(* IEC 61131-3 sources: repolevel_ST_code_completion/dataset/project_code/卷绕机/FUN, 4 files *)

(* ---- FB_DualAxisEmergencyStop.st ---- *)
FUNCTION_BLOCK FB_DualAxisEmergencyStop
VAR_IN_OUT
	AxisM			:	AXIS_REF_SM3;		// 主轴引用
	AxisS			:	AXIS_REF_SM3;		// 从轴引用
END_VAR
VAR_INPUT
	bExecute		:	BOOL;				// 执行紧急停止
	rDeceleration	:	LREAL := 36000;		// 减速度
END_VAR
VAR_OUTPUT
	bDone			:	BOOL;				// 停止完成
	bBusy			:	BOOL;				// 停止进行中
	bError			:	BOOL;				// 错误标志
END_VAR
VAR
	fbHaltM			:	MC_Halt;			// 主轴停止功能块
	fbHaltS			:	MC_Halt;			// 从轴停止功能块
	fbRtrigExecute	:	R_TRIG;				// 执行上升沿检测
	nState			:	BYTE;				// 内部状态机
END_VAR

fbRtrigExecute(CLK := bExecute);

CASE nState OF
	0: // 空闲/初始化
		bDone := FALSE;
		bBusy := FALSE;
		bError := FALSE;
		fbHaltM(Axis := AxisM, Execute := FALSE);
		fbHaltS(Axis := AxisS, Execute := FALSE);

		IF fbRtrigExecute.Q THEN
			nState := 1;
			bBusy := TRUE;
		END_IF

	1: // 执行双轴停止
		fbHaltM(
			Axis := AxisM,
			Execute := TRUE,
			Deceleration := rDeceleration
		);

		fbHaltS(
			Axis := AxisS,
			Execute := TRUE,
			Deceleration := rDeceleration
		);

		// 等待两轴都停止完成
		IF fbHaltM.Done AND fbHaltS.Done THEN
			nState := 2;
		END_IF

		// 错误检查
		IF fbHaltM.Error OR fbHaltS.Error THEN
			bError := TRUE;
			nState := 100;
		END_IF

	2: // 复位Halt功能块
		fbHaltM(Axis := AxisM, Execute := FALSE);
		fbHaltS(Axis := AxisS, Execute := FALSE);
		nState := 3;

	3: // 完成
		bDone := TRUE;
		bBusy := FALSE;
		nState := 0;

	100: // 错误状态
		bError := TRUE;
		bBusy := FALSE;
		fbHaltM(Execute := FALSE);
		fbHaltS(Execute := FALSE);
		// 等待bExecute复位
		IF NOT bExecute THEN
			nState := 0;
		END_IF
END_CASE

(* ---- FB_DualAxisPower.st ---- *)
FUNCTION_BLOCK FB_DualAxisPower
VAR_IN_OUT
	AxisM		:	AXIS_REF_SM3;		// 主轴引用
	AxisS		:	AXIS_REF_SM3;		// 从轴引用
END_VAR
VAR_INPUT
	bPowerOn	:	BOOL;				// 电源使能信号
END_VAR
VAR_OUTPUT
	bReady		:	BOOL;				// 两轴都准备就绪
	bAxisMReady	:	BOOL;				// 主轴准备状态
	bAxisSReady	:	BOOL;				// 从轴准备状态
	bError		:	BOOL;				// 错误标志
END_VAR
VAR
	fbPowerM	:	SM3_Basic.MC_Power;	// 主轴电源控制
	fbPowerS	:	SM3_Basic.MC_Power;	// 从轴电源控制
END_VAR

// 主轴电源控制
fbPowerM(
	Axis := AxisM,
	Enable := TRUE,
	bRegulatorOn := bPowerOn,
	bDriveStart := bPowerOn
);

// 从轴电源控制
fbPowerS(
	Axis := AxisS,
	Enable := TRUE,
	bRegulatorOn := bPowerOn,
	bDriveStart := bPowerOn
);

// 更新输出状态
bAxisMReady := fbPowerM.Status;
bAxisSReady := fbPowerS.Status;
bReady := fbPowerM.Status AND fbPowerS.Status;

// 错误处理
bError := fbPowerM.Error OR fbPowerS.Error;

(* ---- SeekHome.st ---- *)
FUNCTION_BLOCK SeekHome
VAR_IN_OUT
	_Axis	:	AXIS_REF_SM3;
END_VAR
VAR_INPUT
	_xHome	:	BOOL;
	_xAbort	:	BOOL;
	_nHomeMode	:	HomeMode;
	_fFastHomeVel	:	LREAL;
	_fSlowHomeVel	:	LREAL;
	_fHomeAcc		:	LREAL;
	_fHomeDec		:	LREAL;
	_fHomePos		:	LREAL;
	_xReferenceSwitch	:	BOOL;//typically is true
	_nDirection	:	MC_DIRECTION;
	_xIndexPulse	:	BOOL;
END_VAR
VAR_OUTPUT
	_xBusy	:	BOOL;
	_xDone	:	BOOL;
	_xErr	:	BOOL;
	_iErrId	:	DINT;
END_VAR
VAR
	_fbMoveVel	:	MC_MoveVelocity;
	_fbMoveAbs	:	MC_MoveAbsolute;
	_fbHalt		:	MC_Halt;
	_fbSetPos	:	MC_SetPosition;
	_fbRtrig		:	R_TRIG;
	_fbFtrig		:	F_TRIG;
	_nBDirection	:	MC_DIRECTION;
	_fTempPos		:	LREAL;
	_nState		:	USINT;
	fbRtrig	:	R_TRIG;
END_VAR

//check left / arrive the ReferenceSwitch
_fbRtrig(CLK := _xReferenceSwitch);
_fbFtrig(CLK := _xReferenceSwitch);
fbRtrig(CLK := _xHome);

IF NOT _xHome THEN
	_fbMoveVel(Axis := _Axis,Execute := FALSE);
	_fbMoveAbs(Axis := _Axis,Execute := FALSE);
	_fbHalt(Axis := _Axis,Execute := FALSE);
	_fbSetPos(Axis := _Axis,Execute := FALSE);
	_xDone := FALSE;
	_xErr := FALSE;
END_IF

CASE _nState OF
	0:
		IF fbRtrig.Q THEN
			_xBusy := TRUE;
			_xDone := FALSE;
			_xErr := FALSE;
			_iErrId := 0;

			CASE _nDirection OF //cal which is the invert direction
				MC_DIRECTION.positive:
					_nBDirection := MC_DIRECTION.negative;
				MC_DIRECTION.negative:
					_nBDirection := MC_DIRECTION.positive;
				ELSE
					_xErr := TRUE;
			END_CASE

			CASE _nHomeMode OF
				HomeMode.FAST_ZERO:
					_fTempPos := 0;
					_nState := 21;
				HomeMode.FAST_BSLOW_STOP_S:
					_nState := 1;
				HomeMode.FAST_SLOW_STOP_S:
					_nState := 11;
				HomeMode.FAST_BSLOW_I_STOP_S:
					_nState := 31;
				HomeMode.FAST_SLOW_I_STOP_S:
					_nState := 41;
			END_CASE
		END_IF
	50:
		_fbMoveAbs(Execute := TRUE,Axis := _Axis,Position := _fTempPos,Velocity := _fSlowHomeVel,Acceleration := _fHomeAcc,Deceleration := _fHomeDec);
		IF _fbMoveAbs.Done THEN
			_fbMoveAbs(Execute := FALSE,Axis := _Axis);
			_nState := 100;
		END_IF
		IF _fbMoveAbs.Error THEN//meet error
			_nState := 200;
			_iErrId := _fbMoveAbs.ErrorID;
		END_IF
	100:
		_fbSetPos(Execute := TRUE,Axis := _Axis,Position := _fHomePos,Mode := FALSE);//set absolute position
		IF _fbSetPos.Done THEN
			_fbSetPos(Execute := FALSE,Axis := _Axis);
			_xDone := TRUE;
			_xBusy := FALSE;
			_nState := 0;
		END_IF
		IF _fbSetPos.Error THEN//meet error
			_iErrId := _fbSetPos.ErrorID;
			_nState := 200;
		END_IF
	200:
		_xErr := TRUE;
		_xBusy := FALSE;
		_nState := 0;
END_CASE

FAST_ZERO();
FAST_BSLOW_STOP_S();
FAST_SLOW_STOP_S();
FAST_BSLOW_I_STOP_S();
FAST_SLOW_I_STOP_S();

(* ---- StarWork.st ---- *)
FUNCTION_BLOCK StarWork
VAR_IN_OUT
	_AxisW	:	AXIS_REF_SM3;
	_AxisU	:	AXIS_REF_SM3;
	_AxisV	:	AXIS_REF_SM3;
END_VAR
VAR_INPUT
	_bStart	:	BOOL;
	_bStop	:	BOOL;
	_bCheckR	:	BOOL;
	_bFFlag		:	BOOL;
	_lD		:	LREAL;
	_lTk	:	LREAL;
	_lVel	:	LREAL;
	_nDirection	:	MC_DIRECTION;
END_VAR
VAR_OUTPUT
	_xDone	:	BOOL;
	_xErr	:	BOOL;
	_iErrId	:	DINT;
END_VAR
VAR
	_fbAxisWMoveRel	:	SM3_Basic.MC_MoveRelative;
	_fbAxisUMoveRel	:	SM3_Basic.MC_MoveRelative;
	_fbAxisWMoveVelocity: SM3_Basic.MC_MoveVelocity;
	_fbAxisUMoveVelocity: SM3_Basic.MC_MoveVelocity;
	_fbAxisWFollowVelocity:SM3_Basic.SMC_FollowVelocity;
	_fbAxisUFollowVelocity:SM3_Basic.SMC_FollowVelocity;
	_fbHaltAxisW		:	MC_Halt;
	_fbHaltAxisU		:	MC_Halt;
	_fbStartRtrig	:	R_TRIG;
	_fbStopRtrig		:	R_TRIG;
	_fbCheckRtrig		:	R_TRIG;
	_AxisPID:Util.PID_FIXCYCLE;

	AxisWVel:LREAL;
	AxisUVel:LREAL;
	AxisWOldPoint,AxisWNewPoint:LREAL;
	AxisUOldPoint,AxisUNewPoint:LREAL;
	AxisVOldPoint,AxisVNewPoint:LREAL;

	_iStatus :	INT;
	Hold,Hnew:LREAL;
	Lold,Lnew:LREAL;
	Wr,Ur:LREAL;//半径
	PIDOut: REAL;
END_VAR

CASE _iStatus OF
	3:
		_fbAxisWMoveVelocity(Axis:=_AxisW,Execute:=TRUE,Velocity:=20,Acceleration:=3600,Deceleration:=3600,Direction:=-1);
		IF _AxisV.fActPosition>=211 THEN
			_fbAxisWMoveVelocity(Axis:=_AxisW,Execute:=FALSE);
			_fbHaltAxisW(Axis:=_AxisW,Execute:=FALSE,Deceleration:=3600);
			_iStatus:=4;
		END_IF
	4:
		_fbHaltAxisW(Axis:=_AxisW,Deceleration:=3600,Execute:=TRUE);
		IF _fbHaltAxisW.Done THEN
			_iStatus:=5;
		END_IF

	5://半径测量初始化
	Hold:=_AxisV.fActPosition;
	_fbCheckRtrig(CLK:=_bCheckR);
	IF _fbCheckRtrig.Q THEN
		_fbAxisWMoveRel(Axis:=_AxisW,Execute:=FALSE);
		_fbAxisUMoveRel(Axis:=_AxisU,Execute:=FALSE);
		_iStatus:=6;
	END_IF
		6:
		Hold:=_AxisV.fActPosition;
		_iStatus:=7;
	7:
		_fbAxisUMoveRel(Axis:=_AxisU,Execute:=TRUE,Distance:=360,Velocity:=10,Deceleration:=3600,Acceleration:=3600);
		IF _fbAxisUMoveRel.Done THEN
			Hnew:=_AxisV.fActPosition;
			_fbAxisUMoveRel(Axis:=_AxisU,Execute:=FALSE);
			_iStatus:=8;
		END_IF
	8:
		Ur:=ABS(SQRT(EXPT(_lD,2)+EXPT(Hnew+31,2))-SQRT(EXPT(_lD,2)+EXPT(Hold+31,2)))/SMC_PI+_lTk;
		Hold:=_AxisV.fActPosition;
		_iStatus:=9;

	9://半径测量
		_fbAxisWMoveRel(Axis:=_AxisW,Execute:=TRUE,Distance:=-360,Velocity:=10,Acceleration:=3600,Deceleration:=3600);
		IF _fbAxisWMoveRel.Done THEN
			Hnew:=_AxisV.fActPosition;
			_fbAxisWMoveRel(Axis:=_AxisW,Execute:=FALSE);
			_iStatus:=10;
		END_IF
	10:
		Wr:=ABS(SQRT(EXPT(_lD,2)+EXPT(Hnew+31,2))-SQRT(EXPT(_lD,2)+EXPT(Hold+31,2)))/SMC_PI+_lTk;
		   _iStatus:=11;
	11:
		AxisWVel:=_lVel;
		AxisUVel:=-1*AxisWVel*Wr/Ur;
		AxisWOldPoint:=_AxisW.fActPosition;
		AxisUOldPoint:=_AxisU.fActPosition;
		AxisVOldPoint:=_AxisV.fActPosition;
		_iStatus:=12;

	12:
		IF AxisWOldPoint>_AxisW.fActPosition THEN
			AxisWVel:=AxisWVel+AxisWVel*_lTk/(Wr-_lTk);
		END_IF
		IF AxisUOldPoint>_AxisU.fActPosition THEN
			AxisUVel:=AxisUVel-AxisUVel*_lTk/(Ur+_lTk);
		END_IF
		_fbAxisWFollowVelocity(Axis:=_AxisW,bExecute:=TRUE,fSetVelocity:=AxisWVel);
		_fbAxisUFollowVelocity(Axis:=_AxisU,bExecute:=TRUE,fSetVelocity:=AxisUVel);
		_AxisPID(ACTUAL:=AxisV.fActPosition,SET_POINT:=AxisVOldPoint,KP:=0.05,TN:=5,TV:=0,CYCLE:=0.004,Y=>PIDOut);
		AxisUVel:=AxisUVel-PIDOut;
		AxisWOldPoint:=_AxisW.fActPosition;
		AxisUOldPoint:=_AxisU.fActPosition;
END_CASE
